// TwinCAT 3 PLC project Untitled1
// ProgramVersion: 3.1.4022.7
// libraries:
//   L2SI Vacuum Library
//   LCLS General, * (SLAC)
//   PMPS, * (SLAC - LCLS)
//   Tc2_Standard, * (Beckhoff Automation GmbH)
//   Tc2_System, * (Beckhoff Automation GmbH)
//   Tc2_Utilities, * (Beckhoff Automation GmbH)
//   Tc3_Module, * (Beckhoff Automation GmbH)
// project tree:
//   DUTs/ DUT_EpicsMotorMSTA.TcDUT, DUT_SourceDataStore.TcDUT, FB_DestinationDataStore.TcPOU, FB_EpicsMotorMonitor.TcPOU, FB_EpicsCentroidMonitor.TcPOU, FB_RangeComparison.TcPOU, FB_ShutterSafety.TcPOU
//   GVLs/ GVL_BTPS.TcGVL, GVL_BTPS_Constants.TcGVL, GVL_BTPS_Retain.TcGVL
//   / PlcTask.TcTTO
//   POUs/ F_IsValveReady.TcPOU, MAIN.TcPOU, PRG_SavePeristentVariables.TcPOU
// real-time tasks:
//   TASK PlcTask: cycle T#10ms, priority 20, ADS port 350

CONFIGURATION Untitled1
    RESOURCE PLC ON TwinCAT3
        TASK PlcTask(INTERVAL := T#10ms, PRIORITY := 20);
        PROGRAM MAIN WITH PlcTask : MAIN;
    END_RESOURCE
END_CONFIGURATION

// ---- DUTs/DUT_EpicsMotorMSTA.TcDUT
TYPE DUT_EpicsMotorMSTA :
STRUCT

    (* DIRECTION: last raw direction; (0:Negative, 1:Positive) *)
    bPositiveDirection : BIT;
    (* DONE: motion is complete. *)
    bDone : BIT;
    (* PLUS_LS: plus limit switch has been hit. *)
    bPlusLimitSwitch : BIT;
    (* HOMELS: state of the home limit switch. *)
    bHomeLimitSwitch : BIT;
    (* Unused *)
    bUnused0 : BIT;
    (* POSITION: closed-loop position control is enabled. *)
    bClosedLoop : BIT;
    (* SLIP_STALL: Slip/Stall detected (eg. fatal following error) *)
    bSlipStall : BIT;
    (* HOME: if at home position. *)
    bHome : BIT;
    (* PRESENT: encoder is present. *)
    bEncoderPresent : BIT;
    (* PROBLEM: driver stopped polling, or hardware problem *)
    bHardwareProblem : BIT;
    (* MOVING: non-zero velocity present. *)
    bMoving : BIT;
    (* GAIN_SUPPORT: motor supports closed-loop position control. *)
    bGainSupport : BIT;
    (* COMM_ERR: Controller communication error. *)
    bCommError : BIT;
    (* MINUS_LS: minus limit switch has been hit. *)
    bMinusLimitSwitch : BIT;
    (* HOMED: the motor has been homed. *)
    bHomed : BIT;

END_STRUCT
END_TYPE

// ---- DUTs/DUT_SourceDataStore.TcDUT
TYPE DUT_SourceDataStore :
STRUCT
    {attribute 'pytmc' := 'pv: Name; io: input'}
    sName : STRING;
    {attribute 'pytmc' := 'pv: Valve'}
    fbSourceValve : REFERENCE TO FB_VGC;
    {attribute 'pytmc' := '
        pv: Valid
        io: input
        field: ZNAM Data Invalid
        field: ONAM Data Valid
        field: ZSV MAJOR
        field: OSV NO_ALARM
    '}
    bDataValid : BOOL;

    {attribute 'pytmc' := '
        pv: EntryValveReady
        io: input
        field: ZNAM Not ready
        field: ONAM Ready
        field: ZSV MAJOR
        field: OSV NO_ALARM
    '}
    bEntryValveReady : BOOL;

    {attribute 'pytmc' := '
        pv: ChecksOK
        io: input
        field: ZNAM Failed
        field: ONAM Passed
        field: ZSV MAJOR
        field: OSV NO_ALARM
    '}
    bChecksOK : BOOL;

    {attribute 'pytmc' := 'pv: Linear'}
    fbLinear : FB_RangeComparison;
    {attribute 'pytmc' := 'pv: Rotary'}
    fbRotary : FB_RangeComparison;
    {attribute 'pytmc' := 'pv: Goniometer'}
    fbGoniometer : FB_RangeComparison;
    {attribute 'pytmc' := 'pv: NFCenterX'}
    fbNFCentroidX : FB_RangeComparison;
    {attribute 'pytmc' := 'pv: NFCenterY'}
    fbNFCentroidY : FB_RangeComparison;
    {attribute 'pytmc' := 'pv: FFCenterX'}
    fbFFCentroidX : FB_RangeComparison;
    {attribute 'pytmc' := 'pv: FFCenterY'}
    fbFFCentroidY : FB_RangeComparison;

END_STRUCT
END_TYPE

// ---- GVLs/GVL_BTPS.TcGVL
{attribute 'qualified_only'}
VAR_GLOBAL
    (*
    Motor - Linear
        LAS:BTS:MCS2:01:m1 (ioc-las-bts-mcs1, las_bts_mcs2_01_m1)
        LAS:BTS:MCS2:01:m4 (ioc-las-bts-mcs1, las_bts_mcs2_01_m4)
        LAS:BTS:MCS2:01:m7 (ioc-las-bts-mcs1, las_bts_mcs2_01_m7)
    *)
    {attribute 'pytmc' := '
        pv: @(BTPS):Chk:B1Lin
        link: @(SIM)LAS:BTS:MCS2:01:m1
    '}
    fbBay1Linear : FB_EpicsMotorMonitor;
    {attribute 'pytmc' := '
        pv: @(BTPS):Chk:B3Lin
        link: @(SIM)LAS:BTS:MCS2:01:m4
    '}
    fbBay3Linear : FB_EpicsMotorMonitor;
    {attribute 'pytmc' := '
        pv: @(BTPS):Chk:B4Lin
        link: @(SIM)LAS:BTS:MCS2:01:m7
    '}
    fbBay4Linear : FB_EpicsMotorMonitor;

    (*
        Motor - Rotary
            LAS:BTS:MCS2:01:m2 (ioc-las-bts-mcs1, las_bts_mcs2_01_m2)
            LAS:BTS:MCS2:01:m6 (ioc-las-bts-mcs1, las_bts_mcs2_01_m6)
            LAS:BTS:MCS2:01:m8 (ioc-las-bts-mcs1, las_bts_mcs2_01_m8)
    *)
    {attribute 'pytmc' := '
        pv: @(BTPS):Chk:B1Rot
        link: @(SIM)LAS:BTS:MCS2:01:m2
    '}
    fbBay1Rotary : FB_EpicsMotorMonitor;
    {attribute 'pytmc' := '
        pv: @(BTPS):Chk:B3Rot
        link: @(SIM)LAS:BTS:MCS2:01:m6
    '}
    fbBay3Rotary : FB_EpicsMotorMonitor;
    {attribute 'pytmc' := '
        pv: @(BTPS):Chk:B4Rot
        link: @(SIM)LAS:BTS:MCS2:01:m8
    '}
    fbBay4Rotary : FB_EpicsMotorMonitor;

    (*
        Motor - Goniometer
            LAS:BTS:MCS2:01:m3 (ioc-las-bts-mcs1, las_bts_mcs2_01_m3)
            LAS:BTS:MCS2:01:m5 (ioc-las-bts-mcs1, las_bts_mcs2_01_m5)
            LAS:BTS:MCS2:01:m9 (ioc-las-bts-mcs1, las_bts_mcs2_01_m9)
    *)
    {attribute 'pytmc' := '
        pv: @(BTPS):Chk:B1Gon
        link: @(SIM)LAS:BTS:MCS2:01:m3
    '}
    fbBay1Goniometer : FB_EpicsMotorMonitor;
    {attribute 'pytmc' := '
        pv: @(BTPS):Chk:B3Gon
        link: @(SIM)LAS:BTS:MCS2:01:m5
    '}
    fbBay3Goniometer : FB_EpicsMotorMonitor;
    {attribute 'pytmc' := '
        pv: @(BTPS):Chk:B4Gon
        link: @(SIM)LAS:BTS:MCS2:01:m9
    '}
    fbBay4Goniometer : FB_EpicsMotorMonitor;

    (* Near field camera stats plugins, per bay *)
    {attribute 'pytmc' := '
        pv: @(BTPS):Chk:NF1
        link: @(SIM)LAS:LHN:BAY1:CAM:01:Stats2:
    '}
    fbBay1NearFieldCamStats : FB_EpicsCentroidMonitor;

    {attribute 'pytmc' := '
        pv: @(BTPS):Chk:NF3
        link: @(SIM)LAS:LHN:BAY3:CAM:01:Stats2:
    '}
    fbBay3NearFieldCamStats : FB_EpicsCentroidMonitor;

    {attribute 'pytmc' := '
        pv: @(BTPS):Chk:NF4
        link: @(SIM)LAS:LHN:BAY4:CAM:01:Stats2:
    '}
    fbBay4NearFieldCamStats : FB_EpicsCentroidMonitor;

    (* Far-field camera stats plugins, per bay *)
    {attribute 'pytmc' := '
        pv: @(BTPS):Chk:FF1
        link: @(SIM)LAS:LHN:BAY1:CAM:02:Stats2:
    '}
    fbBay1FarFieldCamStats : FB_EpicsCentroidMonitor;

    {attribute 'pytmc' := '
        pv: @(BTPS):Chk:FF3
        link: @(SIM)LAS:LHN:BAY3:CAM:02:Stats2:
    '}
    fbBay3FarFieldCamStats : FB_EpicsCentroidMonitor;

    {attribute 'pytmc' := '
        pv: @(BTPS):Chk:FF4
        link: @(SIM)LAS:LHN:BAY4:CAM:02:Stats2:
    '}
    fbBay4FarFieldCamStats : FB_EpicsCentroidMonitor;

    (* Temporary valves for testing *)
    fbBay1SourceValve : FB_VGC;
    fbBay3SourceValve : FB_VGC;
    fbBay4SourceValve : FB_VGC;
    fbDestinationValves : ARRAY [1..GVL_BTPS_Constants.nDestinations] OF FB_VGC;

    {attribute 'pytmc' := 'pv: @(BTPS):Shutter:01'}
    fbShutterSafety1 : FB_ShutterSafety;
    {attribute 'pytmc' := 'pv: @(BTPS):Shutter:03'}
    fbShutterSafety3 : FB_ShutterSafety;
    {attribute 'pytmc' := 'pv: @(BTPS):Shutter:04'}
    fbShutterSafety4 : FB_ShutterSafety;

    {attribute 'pytmc' := 'pv: @(BTPS):DEST'}
    fbDestinations : ARRAY [1..GVL_BTPS_Constants.nDestinations] OF FB_DestinationDataStore;

END_VAR

// ---- GVLs/GVL_BTPS_Constants.TcGVL
{attribute 'qualified_only'}
VAR_GLOBAL CONSTANT
    nSources : UINT := 4;
    (* Destinations

        LTLHN:LD8:VGC:01 (ioc-las-bts) - TMO - IP1
        LTLHN:LD10:VGC:01 (ioc-las-bts) - TMO - IP2
        LTLHN:LD2:VGC:01 (ioc-las-bts) - TMO - IP3

        LTLHN:LD6:VGC:01 (ioc-las-bts) - RIX - qRIXS
        LTLHN:LD4:VGC:01 (ioc-las-bts) - RIX - ChemRIXS
        LTLHN:LD14:VGC:01 (ioc-las-bts) - XPP

        LTLHN:LD9:VGC:01 (ioc-las-bts) - Laser Lab

    *)
    nDestinations: UINT := 7;
END_VAR

// ---- GVLs/GVL_BTPS_Retain.TcGVL
{attribute 'qualified_only'}
VAR_GLOBAL PERSISTENT

    {attribute 'pytmc' := '
        pv: @(BTPS):Config:MaxFrameTime
        field: DESC Maximum delay from frame to frame
        field: EGU sec
    '}
    fMaximumFrameTime : LREAL := 5.0;

    {attribute 'pytmc' := '
        pv: @(BTPS):Config:MinCentroidChange
        field: DESC Minimum centroid change to be considered valid
        field: EGU px
    '}
    fMinCentroidChange : LREAL := 0.05;

END_VAR

// ---- POUs/MAIN.TcPOU
PROGRAM MAIN
VAR

    (* TODO NOTES *)
    (*

    1. Disable FP exceptions for the plc task

    *)
END_VAR

GVL_BTPS.fbBay1Linear(bEnable:=TRUE);
GVL_BTPS.fbBay3Linear(bEnable:=TRUE);
GVL_BTPS.fbBay4Linear(bEnable:=TRUE);

GVL_BTPS.fbBay1Rotary(bEnable:=TRUE);
GVL_BTPS.fbBay3Rotary(bEnable:=TRUE);
GVL_BTPS.fbBay4Rotary(bEnable:=TRUE);

GVL_BTPS.fbBay1Goniometer(bEnable:=TRUE);
GVL_BTPS.fbBay3Goniometer(bEnable:=TRUE);
GVL_BTPS.fbBay4Goniometer(bEnable:=TRUE);

GVL_BTPS.fbBay1NearFieldCamStats(bEnable:=TRUE, fMaximumFrameTime:=GVL_BTPS_Retain.fMaximumFrameTime, fMinimumChange:=GVL_BTPS_Retain.fMinCentroidChange);
GVL_BTPS.fbBay3NearFieldCamStats(bEnable:=TRUE, fMaximumFrameTime:=GVL_BTPS_Retain.fMaximumFrameTime, fMinimumChange:=GVL_BTPS_Retain.fMinCentroidChange);
GVL_BTPS.fbBay4NearFieldCamStats(bEnable:=TRUE, fMaximumFrameTime:=GVL_BTPS_Retain.fMaximumFrameTime, fMinimumChange:=GVL_BTPS_Retain.fMinCentroidChange);

GVL_BTPS.fbBay1FarFieldCamStats(bEnable:=TRUE, fMaximumFrameTime:=GVL_BTPS_Retain.fMaximumFrameTime, fMinimumChange:=GVL_BTPS_Retain.fMinCentroidChange);
GVL_BTPS.fbBay3FarFieldCamStats(bEnable:=TRUE, fMaximumFrameTime:=GVL_BTPS_Retain.fMaximumFrameTime, fMinimumChange:=GVL_BTPS_Retain.fMinCentroidChange);
GVL_BTPS.fbBay4FarFieldCamStats(bEnable:=TRUE, fMaximumFrameTime:=GVL_BTPS_Retain.fMaximumFrameTime, fMinimumChange:=GVL_BTPS_Retain.fMinCentroidChange);

GVL_BTPS.fbDestinations[1](sName:='TMO IP1', fbDestinationValve:=GVL_BTPS.fbDestinationValves[1]);
GVL_BTPS.fbDestinations[2](sName:='TMO IP2', fbDestinationValve:=GVL_BTPS.fbDestinationValves[2]);
GVL_BTPS.fbDestinations[3](sName:='TMO IP3', fbDestinationValve:=GVL_BTPS.fbDestinationValves[3]);
GVL_BTPS.fbDestinations[4](sName:='RIX qRIXS', fbDestinationValve:=GVL_BTPS.fbDestinationValves[4]);
GVL_BTPS.fbDestinations[5](sName:='RIX ChemRIXS', fbDestinationValve:=GVL_BTPS.fbDestinationValves[5]);
GVL_BTPS.fbDestinations[6](sName:='XPP', fbDestinationValve:=GVL_BTPS.fbDestinationValves[6]);
GVL_BTPS.fbDestinations[7](sName:='Laser Lab', fbDestinationValve:=GVL_BTPS.fbDestinationValves[7]);

(* Shutter safety evaluation should always come at the end. *)
GVL_BTPS.fbShutterSafety1(nSourceIndex:=1);
// GVL_BTPS.fbShutterSafety2(nIndex:=2);
GVL_BTPS.fbShutterSafety3(nSourceIndex:=3);
GVL_BTPS.fbShutterSafety4(nSourceIndex:=4);

PRG_SavePeristentVariables();

END_PROGRAM

// ---- POUs/PRG_SavePeristentVariables.TcPOU
PROGRAM PRG_SavePeristentVariables
VAR
    fbWritePersistentData: FB_WritePersistentData;
    tonStart : TON;
    tonInterval : TON;
END_VAR

tonInterval(
    IN:=TRUE,
    PT:=T#1ms (* Write 1ms after startup of the PLC *)

);

tonStart(
    IN:=tonStart.Q AND NOT fbWritePersistentData.BUSY,
    PT:=T#1m (* Write every minute *)
);

fbWritePersistentData(
    NETID:='', (* This PLC *)
    PORT:=851, (* Application port! *)
    TMOUT:=T#10s,  (* Maximum time before considering this a failure *)
    START:=tonStart.Q OR tonInterval.Q (* Start with tonStart goes high or periodically *)
);

END_PROGRAM

// ---- DUTs/FB_EpicsMotorMonitor.TcPOU
(*
    EPICS Motor Record Monitoring tool

    Requires a "link" pragma to specify the motor record prefix.

*)
FUNCTION_BLOCK FB_EpicsMotorMonitor
VAR_INPUT
    bEnable : BOOL := TRUE;
END_VAR
VAR_OUTPUT
    bIsMoving : BOOL;
    fPosition : LREAL;
    nMSTA_Raw : UINT;
    stMSTA : DUT_EpicsMotorMSTA;
    bValid : BOOL;
END_VAR
VAR
    {attribute 'pytmc' := '
        pv: RBV_
        link: .RBV
    '}
    fbRBVCheck : FB_LREALFromEPICS;

    {attribute 'pytmc' := '
        pv: Dmov_
        link: .DMOV
    '}
    fbMovingCheck : FB_LREALFromEPICS;

    {attribute 'pytmc' := '
        pv: Msta_
        link: .MSTA
    '}
    fbMotorStatusCheck : FB_LREALFromEPICS;
END_VAR

IF NOT bEnable THEN
    bValid := FALSE;
    RETURN;
END_IF

fbRBVCheck();
fbMovingCheck();
fbMotorStatusCheck();
bValid := (
    fbRBVCheck.bValid AND
    fbMovingCheck.bValid AND
    fbMotorStatusCheck.bValid
);
bIsMoving := ABS(fbMovingCheck.fValue) < 1e-5;
fPosition := fbRBVCheck.fValue;

nMSTA_Raw := LREAL_TO_UINT(fbMotorStatusCheck.fValue);
stMSTA.bPositiveDirection := nMSTA_Raw.0;
stMSTA.bDone := nMSTA_Raw.1;
stMSTA.bPlusLimitSwitch := nMSTA_Raw.2;
stMSTA.bHomeLimitSwitch := nMSTA_Raw.3;
stMSTA.bUnused0 := nMSTA_Raw.4;
stMSTA.bClosedLoop := nMSTA_Raw.5;
stMSTA.bSlipStall := nMSTA_Raw.6;
stMSTA.bHome := nMSTA_Raw.7;
stMSTA.bEncoderPresent := nMSTA_Raw.8;
stMSTA.bHardwareProblem := nMSTA_Raw.9;
stMSTA.bMoving := nMSTA_Raw.10;
stMSTA.bGainSupport := nMSTA_Raw.11;
stMSTA.bCommError := nMSTA_Raw.12;
stMSTA.bMinusLimitSwitch := nMSTA_Raw.13;
stMSTA.bHomed := nMSTA_Raw.14;

END_FUNCTION_BLOCK

// ---- DUTs/FB_EpicsCentroidMonitor.TcPOU
(*
    EPICS AreaDetector Stats Plugin Centroid Monitor

    Requires a "link" pragma to specify the full plugin prefix.

*)
FUNCTION_BLOCK FB_EpicsCentroidMonitor
VAR_INPUT
    fMaximumFrameTime : LREAL := 0.2;
    bEnable : BOOL := TRUE;
END_VAR
VAR_OUTPUT
    {attribute 'pytmc' := '
        pv: IsUpdating
        io: input
    '}
    bIsUpdating : BOOL;
    {attribute 'pytmc' := '
        pv: CentroidX
        io: input
    '}
    fCentroidX : LREAL;
    {attribute 'pytmc' := '
        pv: CentroidY
        io: input
    '}
    fCentroidY : LREAL;
    {attribute 'pytmc' := '
        pv: ArrayCount
        io: input
    '}
    nArrayCount : UDINT;
    bValid : BOOL;
    {attribute 'pytmc' := '
        pv: FrameTime
        io: input
        field: DESC Time between frame updates
        field: EGU sec
    '}
    fFrameTime : LREAL;
END_VAR
VAR
    {attribute 'pytmc' := '
        pv: CX_
        link: CentroidX_RBV
    '}
    fbCentroidX : FB_LREALFromEPICS;

    {attribute 'pytmc' := '
        pv: CY_
        link: CentroidY_RBV
    '}
    fbCentroidY : FB_LREALFromEPICS;

    {attribute 'pytmc' := '
        pv: Cnt_
        link: ArrayCounter_RBV
    '}
    fbArrayCounter : FB_LREALFromEPICS;

    // Last array count value
    nLastArrayCount : UDINT;
    // Time of the last frame update
    tLastUpdate: TIME;

    bInit : BOOL;
    // Did we see a frame update yet?
    bSawFrame : BOOL;

END_VAR

IF NOT bEnable THEN
    bValid := FALSE;
    RETURN;
END_IF

IF NOT bInit THEN
    tLastUpdate := TIME();
    fFrameTime := 1000.0;
    bSawFrame := FALSE;
    bInit := TRUE;
END_IF

fbCentroidX();
fbCentroidY();
fbArrayCounter();

bValid := (
    fbCentroidX.bValid AND
    fbCentroidY.bValid AND
    fbArrayCounter.bValid
);

fCentroidX := fbCentroidX.fValue;
fCentroidY := fbCentroidY.fValue;
nArrayCount := LREAL_TO_UDINT(fbArrayCounter.fValue);

IF nArrayCount <> nLastArrayCount THEN
    fFrameTime := TIME_TO_LREAL(TIME() - tLastUpdate) * 0.001; // Milliseconds -> seconds
    tLastUpdate := TIME();
    nLastArrayCount := nArrayCount;
    bSawFrame := TRUE;
END_IF

bIsUpdating := bSawFrame AND (fFrameTime <= GVL_BTPS_Retain.fMaximumFrameTime);

END_FUNCTION_BLOCK

// ---- DUTs/FB_ShutterSafety.TcPOU
FUNCTION_BLOCK FB_ShutterSafety
VAR_INPUT

    {attribute 'pytmc' := '
        pv: LSS:Permission
        io: input
        field: ZNAM No permission
        field: ONAM Permission
    '}
    bLssPermission : BOOL;

    {attribute 'pytmc' := '
        pv: Acknowledge
        io: io
        field: ZNAM FALSE
        field: ONAM TRUE
    '}
    bAcknowledge : BOOL;

    {attribute 'pytmc' := '
        pv: UserOpen
        io: io
        field: ZNAM Close
        field: ONAM Open
    '}
    bUserOpenRequest : BOOL;

    {attribute 'pytmc' := '
        pv: Override
        io: io
        field: ZNAM Normal mode
        field: ONAM Override mode
    '}
    bOverride : BOOL;

    nSourceIndex : UINT;

END_VAR
VAR_OUTPUT

    {attribute 'pytmc' := '
        pv: Safe
        io: input
        field: ZNAM Unsafe
        field: ONAM Safe
    '}
    bSafeToOpen : BOOL;

    {attribute 'pytmc' := '
        pv: Error
        io: input
        field: ZNAM No error
        field: ONAM Error
        field: ZSV NO_ALARM
        field: OSV MAJOR
    '}
    bLatchedError : BOOL;

    {attribute 'pytmc' := '
        pv: LSS:OpenRequest
        io: input
        field: ZNAM Request close
        field: ONAM Request open
    '}
    bOpenSignal : BOOL;

    (* Rising trigger indicator of a new error condition. *)
    rtError : R_TRIG;
    (* Rising trigger indicator of user requesting override. *)
    rtOverrideSet : R_TRIG;
    (* Falling trigger for a 'close shutter' request. *)
    ftCloseRequest : F_TRIG;

END_VAR
VAR

    nDestIndex : UINT;
    bBtpsPermission : BOOL;

END_VAR

bLatchedError R= bAcknowledge;
bAcknowledge := FALSE;

IF nSourceIndex >= 1 AND nSourceIndex <= GVL_BTPS_Constants.nSources THEN
	bBtpsPermission := FALSE;
	FOR nDestIndex := 1 TO GVL_BTPS_Constants.nDestinations DO
		bBtpsPermission := (
			bBtpsPermission OR
			GVL_BTPS.fbDestinations[nDestIndex].stSourceDataStore[nSourceIndex].bChecksOK
		);
	END_FOR
ELSE
    bBtpsPermission := FALSE;
    bLatchedError := TRUE;
END_IF

(* Latch an error if we have no permission. *)
bLatchedError S= NOT bBtpsPermission;
rtError(CLK:=bLatchedError);

(* Reset the user open request on a new error (if not in override mode) *)
bUserOpenRequest R= rtError.Q AND NOT bOverride;

(* If the user requesets a shutter close, clear override mode. *)
ftCloseRequest(CLK:=bUserOpenRequest);
bOverride R= ftCloseRequest.Q;

(* Don't open immediately when in override mode.  Make the user request it. *)
rtOverrideSet(CLK:=bOverride);
bUserOpenRequest R= rtOverrideSet.Q AND NOT bBtpsPermission;

(* Lose permission on a latched error. *)
bBtpsPermission R= bLatchedError;

(* TODO: Where do we get LSS Permission from? *)
// bOverride R= NOT bLssPermission;

(* It's safe to open IF in override mode (user says so!) or we determined it. *)
bSafeToOpen := bOverride OR bBtpsPermission;

(* Only open the shutter if requested and it's safe. *)
bOpenSignal := bSafeToOpen AND bUserOpenRequest;

END_FUNCTION_BLOCK

// ---- DUTs/FB_DestinationDataStore.TcPOU
FUNCTION_BLOCK FB_DestinationDataStore
VAR_INPUT
    {attribute 'pytmc' := 'pv: Name; io: input'}
    sName : STRING;
    {attribute 'pytmc' := 'pv: DestValve'}
    fbDestinationValve : REFERENCE TO FB_VGC;

    {attribute 'pytmc' := '
        pv: ExitValveReady
        io: input
        field: ZNAM Not ready
        field: ONAM Ready
        field: ZSV MAJOR
        field: OSV NO_ALARM
    '}
    bExitValveReady : BOOL;

    {attribute 'pytmc' := 'pv: SRC'}
	stSourceDataStore : ARRAY [1..GVL_BTPS_Constants.nSources] OF DUT_SourceDataStore;
END_VAR
VAR_OUTPUT
    // 
    bDataValid : BOOL;
END_VAR
VAR
    nIndex : UINT;
    stSource: REFERENCE TO DUT_SourceDataStore;
END_VAR

bExitValveReady := F_IsValveReady(fbDestinationValve);

Update(
    stDataSource:=stSourceDataStore[1],
    sName:='Source 1',
    fbSourceValve:=GVL_BTPS.fbBay1SourceValve,
    fbLinear:=GVL_BTPS.fbBay1Linear,
    fbRotary:=GVL_BTPS.fbBay1Rotary,
    fbGoniometer:=GVL_BTPS.fbBay1Goniometer,
    fbNearField:=GVL_BTPS.fbBay1NearFieldCamStats,
    fbFarField:=GVL_BTPS.fbBay1FarFieldCamStats
);

// Future use:
(*
Update(
    stDataSource:=stSourceDataStore2,
    sName:='Source 2',
    fbSourceValve:=GVL_BTPS.fbBay2SourceValve,
    fbLinear:=GVL_BTPS.fbBay2Linear,
    fbRotary:=GVL_BTPS.fbBay2Rotary,
    fbGoniometer:=GVL_BTPS.fbBay2Goniometer,
    fbNearField:=GVL_BTPS.fbBay2NearFieldCamStats,
    fbFarField:=GVL_BTPS.fbBay2FarFieldCamStats
);
*)

Update(
    stDataSource:=stSourceDataStore[3],
    sName:='Source 3',
    fbSourceValve:=GVL_BTPS.fbBay3SourceValve,
    fbLinear:=GVL_BTPS.fbBay3Linear,
    fbRotary:=GVL_BTPS.fbBay3Rotary,
    fbGoniometer:=GVL_BTPS.fbBay3Goniometer,
    fbNearField:=GVL_BTPS.fbBay3NearFieldCamStats,
    fbFarField:=GVL_BTPS.fbBay3FarFieldCamStats
);

Update(
    stDataSource:=stSourceDataStore[4],
    sName:='Source 4',
    fbSourceValve:=GVL_BTPS.fbBay4SourceValve,
    fbLinear:=GVL_BTPS.fbBay4Linear,
    fbRotary:=GVL_BTPS.fbBay4Rotary,
    fbGoniometer:=GVL_BTPS.fbBay4Goniometer,
    fbNearField:=GVL_BTPS.fbBay4NearFieldCamStats,
    fbFarField:=GVL_BTPS.fbBay4FarFieldCamStats
);

METHOD Update : BOOL
VAR_INPUT
    sName : STRING;
END_VAR
VAR_IN_OUT
    // The data source to update
    stDataSource : DUT_SourceDataStore;

    // The source information
    fbSourceValve : FB_VGC;
    fbNearField : FB_EpicsCentroidMonitor;
    fbFarField : FB_EpicsCentroidMonitor;
    fbLinear : FB_EpicsMotorMonitor;
    fbRotary : FB_EpicsMotorMonitor;
    fbGoniometer : FB_EpicsMotorMonitor;

END_VAR
stDataSource.sName := sName;
stDataSource.fbSourceValve REF= fbSourceValve;

stDataSource.bEntryValveReady := F_IsValveReady(fbSourceValve);

(* Update range comparisons with their source values *)
(* Cameras *)
stDataSource.fbNFCentroidX.fValue := fbNearField.fCentroidX;
stDataSource.fbNFCentroidX.bInputValid := fbNearField.bValid AND fbNearField.bIsUpdating;
stDataSource.fbNFCentroidY.fValue := fbNearField.fCentroidY;
stDataSource.fbNFCentroidY.bInputValid := fbNearField.bValid AND fbNearField.bIsUpdating;
stDataSource.fbFFCentroidX.fValue := fbFarField.fCentroidX;
stDataSource.fbFFCentroidX.bInputValid := fbFarField.bValid AND fbFarField.bIsUpdating;
stDataSource.fbFFCentroidY.fValue := fbFarField.fCentroidY;
stDataSource.fbFFCentroidY.bInputValid := fbFarField.bValid AND fbFarField.bIsUpdating;

(* Motors *)
stDataSource.fbLinear.fValue := fbLinear.fPosition;
stDataSource.fbLinear.bInputValid := fbLinear.bValid AND fbLinear.stMSTA.bHomed;
stDataSource.fbRotary.fValue := fbRotary.fPosition;
stDataSource.fbRotary.bInputValid := fbRotary.bValid AND fbRotary.stMSTA.bHomed;
stDataSource.fbGoniometer.fValue := fbGoniometer.fPosition;
stDataSource.fbGoniometer.bInputValid := fbGoniometer.bValid AND fbGoniometer.stMSTA.bHomed;

(* Run the range comparisons *)
stDataSource.fbNFCentroidX();
stDataSource.fbNFCentroidY();
stDataSource.fbFFCentroidX();
stDataSource.fbFFCentroidY();
stDataSource.fbLinear();
stDataSource.fbRotary();
stDataSource.fbGoniometer();

(* Data is valid overall if *all* range comparisons say so *)
stDataSource.bDataValid := (
    stDataSource.fbNFCentroidX.bInputValid AND
    stDataSource.fbNFCentroidY.bInputValid AND
    stDataSource.fbFFCentroidX.bInputValid AND
    stDataSource.fbFFCentroidY.bInputValid AND
    stDataSource.fbLinear.bInputValid AND
    stDataSource.fbRotary.bInputValid AND
    stDataSource.fbGoniometer.bInputValid AND
    TRUE
);

(* Checks only pass if data is valid and all comparisons are true *)
stDataSource.bChecksOK := (
    stDataSource.bDataValid AND
    stDataSource.fbNFCentroidX.bInRange AND
    stDataSource.fbNFCentroidY.bInRange AND
    stDataSource.fbFFCentroidX.bInRange AND
    stDataSource.fbFFCentroidY.bInRange AND
    stDataSource.fbLinear.bInRange AND
    stDataSource.fbRotary.bInRange AND
    stDataSource.fbGoniometer.bInRange AND
    stDataSource.bEntryValveReady AND
    bExitValveReady AND
    TRUE
);
END_METHOD

END_FUNCTION_BLOCK

// ---- POUs/F_IsValveReady.TcPOU
FUNCTION F_IsValveReady : BOOL
VAR_IN_OUT
    fbValve : FB_VGC;
END_VAR
VAR
END_VAR

F_IsValveReady := (
    fbValve.iq_stValve.eState = E_ValvePositionState.OPEN AND
    TRUE (*
        * Placeholder for something else?
        * TODO: Do we check eVGC_State for errors?
        * TODO: Do we care if the laser is used at atmosphere?
    *)
);

END_FUNCTION

// ---- DUTs/FB_RangeComparison.TcPOU
FUNCTION_BLOCK FB_RangeComparison
VAR_INPUT PERSISTENT
    (* The low part of the range. *)
    {attribute 'pytmc' := 'pv: Low'}
    fLow : LREAL;
    (* The high part of the range. *)
    {attribute 'pytmc' := 'pv: High'}
    fHigh : LREAL;
    (* Nominal value for this.  User-facing value. *)
    {attribute 'pytmc' := '
        pv: Nominal
        io: io
        field: DESC Nominal value for setting
    '}
    fNominal : LREAL;
END_VAR
VAR_INPUT
    (* The input value for comparison *)
    {attribute 'pytmc' := 'pv: Value; io: input'}
    fValue : LREAL;
    (* Should the input value be trusted? *)
    {attribute 'pytmc' := '
        pv: Valid
        io: input
        field: ZNAM Data Invalid
        field: ONAM Data Valid
        field: ZSV MAJOR
        field: OSV NO_ALARM
    '}
    bInputValid : BOOL := FALSE;
    (* Are the limits inclusive? *)
    {attribute 'pytmc' := '
        pv: Inclusive
        field: ZNAM Exclusive
        field: ONAM Inclusive
    '}
    bInclusive : BOOL := TRUE;
END_VAR
VAR_OUTPUT
    {attribute 'pytmc' := '
        pv: InRange
        io: input
        field: ZNAM Out of range
        field: ONAM In range
        field: ZSV MAJOR
        field: OSV NO_ALARM
    '}
    bInRange : BOOL;
END_VAR

IF NOT bInputValid OR fHigh < fLow THEN
    bInRange := FALSE;
ELSIF bInclusive THEN
    bInRange := (fValue >= fLow) AND (fValue <= fHigh);
ELSE
    bInRange := (fValue > fLow) AND (fValue < fHigh);
END_IF

END_FUNCTION_BLOCK
